(* PLC project Tc2_Utilities.FB_LicFileCopyFromDongle Demo, tc3-libraries-kb TwinCAT 3.1 *)
(* stored: creationDateTime 2026-05-10T20:00:00, modificationDateTime 2026-05-10T20:00:00 *)

PROGRAM P_Demo_FB_LicFileCopyFromDongle
  VAR
    fbFB_LicFileCopyFromDongle : FB_LicFileCopyFromDongle;  (* Tc2_Utilities.FB_LicFileCopyFromDongle 实例 *)
    arg_sNetIdSrc : T_AmsNetId;  (* VAR_INPUT sNetIdSrc *)
    arg_nPortSrc : UINT;  (* VAR_INPUT nPortSrc *)
    arg_sNetIdDest : T_AmsNetId;  (* VAR_INPUT sNetIdDest *)
    arg_sFileNameSrc : STRING;  (* VAR_INPUT sFileNameSrc *)
    arg_sFilePathNameDest : T_MaxString;  (* VAR_INPUT sFilePathNameDest *)
    arg_pCopyBuff : PVOID;  (* VAR_INPUT pCopyBuff *)
    arg_cbCopyLen : UDINT;  (* VAR_INPUT cbCopyLen *)
    arg_bExecute : BOOL;  (* VAR_INPUT bExecute *)
    arg_dwPassCode : DWORD;  (* VAR_INPUT dwPassCode *)
    arg_tTimeout : TIME;  (* VAR_INPUT tTimeout *)
    out_bBusy : BOOL;  (* VAR_OUTPUT bBusy *)
    out_bError : BOOL;  (* VAR_OUTPUT bError *)
    out_nErrorId : UDINT;  (* VAR_OUTPUT nErrorId *)
  END_VAR

            // ============================================================
// Tc2_Utilities.FB_LicFileCopyFromDongle 演示程序（FB 实例）
// ============================================================
// 验证步骤：
//   1. 引用 Tc2_Utilities（及依赖类型所在库 Tc2_System 等）
//   2. 编译 + 登录
//   3. 按 doc.md 给 arg_* 赋值
//   4. 在线监视 out_* / io_* 输出
// ============================================================

fbFB_LicFileCopyFromDongle(
    sNetIdSrc := arg_sNetIdSrc,
    nPortSrc := arg_nPortSrc,
    sNetIdDest := arg_sNetIdDest,
    sFileNameSrc := arg_sFileNameSrc,
    sFilePathNameDest := arg_sFilePathNameDest,
    pCopyBuff := arg_pCopyBuff,
    cbCopyLen := arg_cbCopyLen,
    bExecute := arg_bExecute,
    dwPassCode := arg_dwPassCode,
    tTimeout := arg_tTimeout,
    bBusy => out_bBusy,
    bError => out_bError,
    nErrorId => out_nErrorId
);

          
END_PROGRAM
